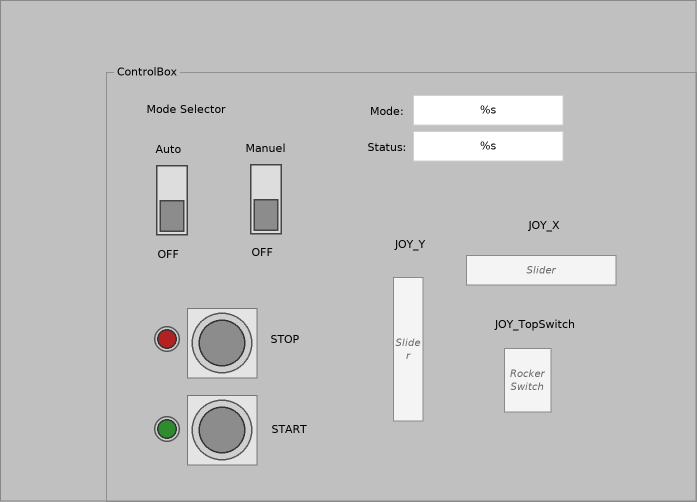
VISUALIZATION VirtualControlBox  // 697x502
    GroupBox (106,64 591x438), "ControlBox"
        PushSwitch (81,244 70x70), variable: VirtualControlBox.bSTOP, behaviour: TOGGLE, style: Switch-PushSwitch-Gray
        PushSwitch (81,331 70x70), variable: VirtualControlBox.bSTART, behaviour: TOGGLE, style: Switch-PushSwitch-Gray
        Slider (360,191 150x30), variable: VirtualControlBox.stJOY.X, scale 0..100
        Slider (287,213 30x144), variable: VirtualControlBox.stJOY.Y, scale -1..1
        RockerSwitch (398,284 47x64), variable: VirtualControlBox.stJOY.Topswitch, behaviour: TOGGLE, style: Switch-RockerSwitch-Gray
        Textfield (307,31 150x30), "%s", text variable: VirtualControlBox.strMode
        Label (378,247 102x27), "JOY_TopSwitch"
        Label (387,148 102x27), "JOY_X"
        Label (253,167 102x27), "JOY_Y"
        Label (233,34 96x27), "Mode:"
        Label (230,70 102x27), "Status:"
        Label (29,32 102x27), "Mode Selector"
        Label (132,352 102x27), "START"
        Label (128,262 102x27), "STOP"
        Lamp1 (46,260 30x30), variable: VirtualControlBox.bSTOP, style: Lamp-Lamp1-Red
        Lamp1 (46,350 30x30), variable: VirtualControlBox.bSTART, style: Lamp-Lamp1-Green
        DipSwitch (31,101 70x70), variable: VirtualControlBox.bAuto, behaviour: TOGGLE, style: Switch-DipSwitch-Gray
        DipSwitch (125,100 70x70), variable: VirtualControlBox.bManual, behaviour: TOGGLE, style: Switch-DipSwitch-Gray
        Label (18,71 89x29), "Auto"
        Label (115,70 89x29), "Manuel"
        Label (18,176 89x29), "OFF"
        Label (112,174 89x29), "OFF"
    Textfield (413,131 150x30), "%s", text variable: VirtualControlBox.strStatus
END_VISUALIZATION

(* stored: Version 1.1.0.1, ProductVersion 3.1.4024.12
   Visu VirtualControlBox: Id {5f34fe80-86f9-499f-8dc6-54b60c760f50} *)
